// TIA Portal V17 export
// export: Created 2025-05-22T06:01:07.2888825Z, ExportSetting WithDefaults, DisplayName Totally Integrated Automation Portal, DisplayVersion V17 Update 8, DisplayName TIA Portal Openness, DisplayVersion V17 Update 8, DisplayName TIA Portal Version Control Interface, DisplayVersion V17, DisplayName SINAMICS Startdrive Advanced, DisplayVersion V17 SP2, DisplayName SINAMICS Startdrive G110M, G120, G120C, G120D, G120P, G115D, DisplayVersion V17 SP2, DisplayName SINAMICS Startdrive G130, G150, S120, S150, SINAMICS MV, S210, DisplayVersion V17 SP2, DisplayName STEP 7 Professional, DisplayVersion V17 Update 8, DisplayName SINUMERIK ONE STEP 7 Toolbox, DisplayVersion V17 Update 12, DisplayName SINUMERIK ONE PLC Basic Program Plus, DisplayVersion V17 Update 12, DisplayName SINUMERIK 840D sl STEP 7 Toolbox, DisplayVersion V17 Update 12, DisplayName STEP 7 Safety, DisplayVersion V17 Update 6, DisplayName WinCC Advanced, DisplayVersion V17 Update 8
DATA_BLOCK "DB1462_SHIELD_AUX_COOLING_ALARMS"   // DB1462
{ S7_Optimized_Access := 'FALSE'; DB_Accessible_From_OPC_UA := 'FALSE' }
VERSION : 0.1
// stored: AutoNumber false, DBAccessibleFromOPCUA false, DBAccessibleFromWebserver true, IsOnlyStoredInLoadMemory false, IsWriteProtectedInAS false
   VAR RETAIN
      UNIT_1 : Struct
         FLOW_VALUE : Real;   // FLOW VALUE
         TEMP_VALUE : Real;   // TEMPERATURE VALUE
         UNIT_01_ALARMS : Struct
            HMI_SETPOINTS : Struct
               FLOW : Struct
                  HIGH_LIMIT_ALM_VALUE : Real;   // HIGH LIMIT ALARM INPUT VALUE
                  LOW_LIMIT_ALM_VALUE : Real;   // LOW LIMIT ALARM INPUT VALUE
                  HIGH_LIMIT_WRN_VALUE : Real;   // HIGH LIMIT WARNING INPUT VALUE
                  LOW_LIMIT_WRN_VALUE : Real;   // LOW LIMIT WARNING INPUT VALUE
               END_STRUCT;
               TEMPERATURE : Struct
                  HIGH_LIMIT_ALM_VALUE : Real;   // HIGH LIMIT ALARM INPUT VALUE
                  LOW_LIMIT_ALM_VALUE : Real;   // LOW LIMIT ALARM INPUT VALUE
                  HIGH_LIMIT_WRN_VALUE : Real;   // HIGH LIMIT WARNING INPUT VALUE
                  LOW_LIMIT_WRN_VALUE : Real;   // LOW LIMIT WARNING INPUT VALUE
               END_STRUCT;
            END_STRUCT;
            ALARMS : Struct
               FLOW : Struct
                  HIGH_LIMIT_ALARM : Bool;   // HIGH LIMIT ALARM ACTIVE
                  LOW_LIMIT_ALARM : Bool;   // LOW LIMIT ALARM ACTIVE
                  HIGH_LIMIT_WARNING : Bool;   // HIGH LIMIT WARNING ACTIVE
                  LOW_LIMIT_WARNING : Bool;   // LOW LIMIT WARNING ACTIVE
               END_STRUCT;
               TEMPERATURE : Struct
                  HIGH_LIMIT_ALARM : Bool;   // HIGH LIMIT ALARM ACTIVE
                  LOW_LIMIT_ALARM : Bool;   // LOW LIMIT ALARM ACTIVE
                  HIGH_LIMIT_WARNING : Bool;   // HIGH LIMIT WARNING ACTIVE
                  LOW_LIMIT_WARNING : Bool;   // LOW LIMIT WARNING ACTIVE
               END_STRUCT;
            END_STRUCT;
         END_STRUCT;
      END_STRUCT;
      UNIT_2 : Struct
         FLOW_VALUE : Real;   // FLOW VALUE
         TEMP_VALUE : Real;   // TEMPERATURE VALUE
         UNIT_02_ALARMS : Struct
            HMI_SETPOINTS : Struct
               FLOW : Struct
                  HIGH_LIMIT_ALM_VALUE : Real;   // HIGH LIMIT ALARM INPUT VALUE
                  LOW_LIMIT_ALM_VALUE : Real;   // LOW LIMIT ALARM INPUT VALUE
                  HIGH_LIMIT_WRN_VALUE : Real;   // HIGH LIMIT WARNING INPUT VALUE
                  LOW_LIMIT_WRN_VALUE : Real;   // LOW LIMIT WARNING INPUT VALUE
               END_STRUCT;
               TEMPERATURE : Struct
                  HIGH_LIMIT_ALM_VALUE : Real;   // HIGH LIMIT ALARM INPUT VALUE
                  LOW_LIMIT_ALM_VALUE : Real;   // LOW LIMIT ALARM INPUT VALUE
                  HIGH_LIMIT_WRN_VALUE : Real;   // HIGH LIMIT WARNING INPUT VALUE
                  LOW_LIMIT_WRN_VALUE : Real;   // LOW LIMIT WARNING INPUT VALUE
               END_STRUCT;
            END_STRUCT;
            ALARMS : Struct
               FLOW : Struct
                  HIGH_LIMIT_ALARM : Bool;   // HIGH LIMIT ALARM ACTIVE
                  LOW_LIMIT_ALARM : Bool;   // LOW LIMIT ALARM ACTIVE
                  HIGH_LIMIT_WARNING : Bool;   // HIGH LIMIT WARNING ACTIVE
                  LOW_LIMIT_WARNING : Bool;   // LOW LIMIT WARNING ACTIVE
               END_STRUCT;
               TEMPERATURE : Struct
                  HIGH_LIMIT_ALARM : Bool;   // HIGH LIMIT ALARM ACTIVE
                  LOW_LIMIT_ALARM : Bool;   // LOW LIMIT ALARM ACTIVE
                  HIGH_LIMIT_WARNING : Bool;   // HIGH LIMIT WARNING ACTIVE
                  LOW_LIMIT_WARNING : Bool;   // LOW LIMIT WARNING ACTIVE
               END_STRUCT;
            END_STRUCT;
         END_STRUCT;
      END_STRUCT;
   END_VAR
BEGIN
END_DATA_BLOCK
